// TwinCAT 3 PLC project Untitled1
// ProgramVersion: 3.1.4024.0
// libraries:
//   Tc2_Standard, * (Beckhoff Automation GmbH)
//   Tc2_System, * (Beckhoff Automation GmbH)
//   Tc3_Module, * (Beckhoff Automation GmbH)
//   VisuDialogs, * (System)
// project tree:
//   / GlobalTextList.TcGTLO, PlcTask.TcTTO, PlcTask1.TcTTO, Visualization Manager.TcVMO (not stored)
//   GVLs/ GVL.TcGVL
//   POUs/ Initialiseren.TcPOU, InvoerEnUitvoer.TcPOU, Simulatie_invoer.TcPOU, Zagen.TcPOU
//   VISUs/ Visualization.TcVIS
// real-time tasks:
//   TASK PlcTask: cycle T#10ms, priority 20, ADS port 350
//   TASK PlcTask1: cycle T#10ms, priority 21, ADS port 351

CONFIGURATION Untitled1
    RESOURCE PLC ON TwinCAT3
        TASK PlcTask(INTERVAL := T#10ms, PRIORITY := 20);
        TASK PlcTask1(INTERVAL := T#10ms, PRIORITY := 21);
        PROGRAM Zagen WITH PlcTask : Zagen;
        PROGRAM InvoerEnUitvoer WITH PlcTask1 : InvoerEnUitvoer;
    END_RESOURCE
END_CONFIGURATION

// ---- GVLs/GVL.TcGVL
{attribute 'qualified_only'}
VAR_GLOBAL
	Power: BOOL := FALSE;
	initialiseren:BOOL := FALSE;
	Initialisatie_voltooid: BOOL := FALSE;
	Status: STRING (INT#30):= 'OFF';
	MotorInvoer: BOOL := 0;
	ZaagLengte: INT :=0;
	HuidigePositieAanvoer: INT := 200;
	StartAanvoer: BOOL;
	AanvoerInPositie: BOOL;
END_VAR

// ---- POUs/Zagen.TcPOU
PROGRAM Zagen
VAR
	MotorUitvoer: BOOL := 0;
	StartZagen: BOOL;
	MotorZagen: BOOL;
	
END_VAR

IF GVL.Power = TRUE THEN 

	
	IF GVL.AanvoerInPositie = TRUE AND StartZagen = TRUE THEN
		MotorZagen :=TRUE;
		GVL.Status:= 'Zaag actief';
		
	END_IF
END_IF

END_PROGRAM

// ---- POUs/InvoerEnUitvoer.TcPOU
PROGRAM InvoerEnUitvoer
VAR

END_VAR

IF gvl.Power = TRUE THEN
		
	IF GVL.Initialisatie_voltooid = FALSE THEN
		Initialiseren();
	END_IF	
	
	IF GVL.Initialisatie_voltooid= TRUE THEN 
			GVL.Status:= 'Voer de zaag lengte in';
	END_IF	

	IF GVL.ZaagLengte >= 0 AND GVL.StartAanvoer = TRUE THEN
		Simulatie_invoer();
	END_IF
		
	IF GVL.ZaagLengte = GVL.HuidigePositieAanvoer AND gvl.ZaagLengte >0 THEN
		gvl.AanvoerInPositie :=TRUE;
		GVL.StartAanvoer:=FALSE;
		GVL.Status:= 'Aanvoer in positie';
	END_IF
	
END_IF

END_PROGRAM

// ---- POUs/Initialiseren.TcPOU
FUNCTION Initialiseren : bool
VAR_INPUT
END_VAR
VAR
END_VAR

IF GVL.HuidigePositieAanvoer >=1 AND GVL.Initialisatie_voltooid = FALSE THEN
		GVL.Status:= 'Initialiseer de machine';
	END_IF

IF GVL.Initialisatie_voltooid = FALSE AND GVL.Initialiseren =TRUE THEN
	Simulatie_Invoer();
		IF gvl.ZaagLengte = gvl.HuidigePositieAanvoer THEN 
			GVL.Initialisatie_voltooid := TRUE;	
			GVL.Initialiseren:=FALSE;	
	END_IF
END_IF

END_FUNCTION

// ---- POUs/Simulatie_invoer.TcPOU
FUNCTION Simulatie_invoer : BOOL
VAR_INPUT
END_VAR
VAR
END_VAR

IF gvl.Power = TRUE THEN
	

	IF GVL.ZaagLengte <= GVL.HuidigePositieAanvoer THEN
		Gvl.MotorInvoer:= TRUE;				
		GVL.HuidigePositieAanvoer := GVL.HuidigePositieAanvoer - 1;
	END_IF;
				
				
	IF GVL.ZaagLengte > GVL.HuidigePositieAanvoer THEN
		Gvl.MotorInvoer:= TRUE;				
		GVL.HuidigePositieAanvoer := GVL.HuidigePositieAanvoer + 1;
	END_IF;
	
	
	IF GVL.ZaagLengte = GVL.HuidigePositieAanvoer THEN
		GVL.MotorInvoer := FALSE;
	END_IF
			
END_IF

END_FUNCTION

// ---- GlobalTextList.TcGTLO
TEXTLIST GlobalTextList
  328 = '%<format string>'
  107 = '%i'
  62 = '%i MAIN.Tekst'
  89 = '%iMAIN.Tekst'
  906 = '%i[MAIN.Tekst]'
  977 = '%MAIN.Tekst'
  479 = '%S'
  169 = '%s'
  410 = 'ggd'
  164 = 'Huidige positie aanvoer'
  363 = 'Initialisatie machine'
  68 = 'Initialiseer de machine'
  209 = 'Initialiseren'
  969 = 'MAIN.Tekst'
  455 = 'Motor aanvoer'
  30 = 'Motor uitvoer'
  607 = 'Start aanvoer'
  5 = 'Start zagen'
  75 = 'Te zagen lengte '
  108 = 'Zaag lengte '
  775 = 'Zaag motor'
END_TEXTLIST

// ---- VISUs/Visualization.TcVIS
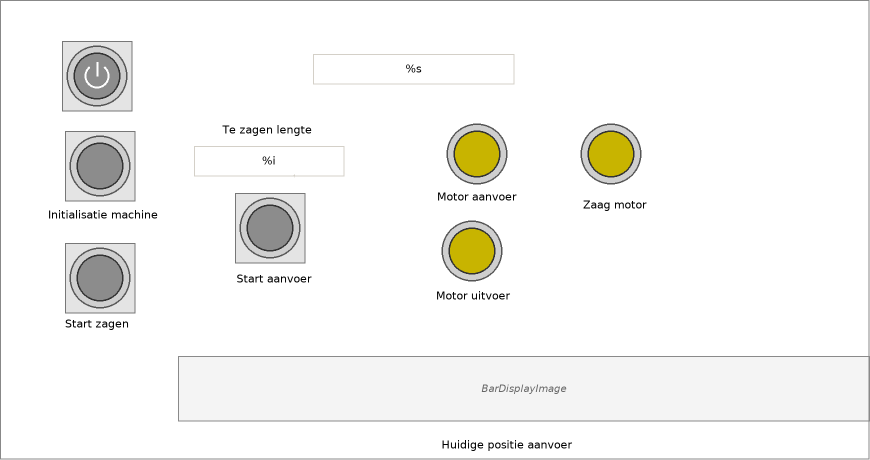
VISUALIZATION Visualization  // 870x460
    PushSwitch (65,131 70x70), variable: GVL.Initialiseren, behaviour: TOGGLE, style: Switch-PushSwitch-Gray
    Textfield (313,54 201x30), "%s", text variable: GVL.Status
    Lamp1 (442,119 70x70), variable: GVL.MotorInvoer, style: Lamp-Lamp1-Yellow
    Lamp1 (437,216 70x70), variable: Zagen.MotorUitvoer, style: Lamp-Lamp1-Yellow
    Label (402,182 150x30), "Motor aanvoer"
    Label (398,281 150x30), "Motor uitvoer"
    Textfield (194,146 150x30), "%i", text variable: GVL.ZaagLengte, invisible if: NOT (GVL.Initialisatie_voltooid)
        OnMouseClick: write GVL.ZaagLengte via VisuDialogs.Numpad, min 1, max 6000
    Label (194,115 150x30), "Te zagen lengte", invisible if: NOT (GVL.Initialisatie_voltooid)
    Label (432,430 150x30), "Huidige positie aanvoer"
    PowerSwitch (62,41 70x70), variable: GVL.Power, behaviour: TOGGLE, style: Switch-PowerSwitch-Gray
    Textfield (294,174 0x3)
    PushSwitch (235,193 70x70), variable: GVL.StartAanvoer, behaviour: TOGGLE, style: Switch-PushSwitch-Gray
    Label (199,264 150x30), "Start aanvoer"
    Label (28,200 150x30), "Initialisatie machine"
    BarDisplayImage (178,356 692x65), value: GVL.HuidigePositieAanvoer, style: BarDisplayImage-Gray, scale format: %.1f, scale 0..2000
    PushSwitch (65,243 70x70), variable: Zagen.StartZagen, behaviour: TOGGLE, style: Switch-PushSwitch-Gray
    Lamp1 (576,119 70x70), variable: Zagen.MotorZagen, style: Lamp-Lamp1-Yellow
    Label (22,309 150x30), "Start zagen"
    Label (540,190 150x30), "Zaag motor"
END_VISUALIZATION
